{attribute 'GeneratedUsingTerminal: EJ1957-0000-0017'}
{attribute addProperty BoxType "EJ1957-0000-0017"}
{attribute addProperty Id "FSOEAT %I*FSOE_BBC930F718"}
{attribute addProperty CRC "2321529592"}
{attribute addProperty Size "18"}
TYPE FSoE_Inputs_8A5FBAF8 :
STRUCT
	{attribute addProperty Name "FSOE"}
	FSOE AT %I* : FSOE_BBC930F7;
END_STRUCT
END_TYPE

(* stored: Version 1.2.0.0, ProductVersion 3.1.4024.9
   DUT FSoE_Inputs_8A5FBAF8: Id {cf906525-b2ed-4273-aefe-03c279faeb10} *)
